//==================================================================================================
//								RJM Maszyny sp. z o.o.
//									13.05.2022
//	Program główny sterujący  
// 	v1.0	|| TC v 3.1.4024.22		|| - pierwsza wersja
//==================================================================================================
PROGRAM MAIN
VAR
	bCzujnik0								: FB_Czujnik_NO;
	bCzujnikMax								: FB_Czujnik_NO;
	fbElektrozawor							: FB_Elektrozawor_5na2_2Cewki;
	fbSilownik								: FB_Silownik_Kontola (fbCzujnikPozycja0 := bCzujnik0, 
																	fbCzujnikPozycjaMax := bCzujnikMax,
																	fbElektrozawor := fbElektrozawor);
	bDoPoczatku: BOOL;
	bDoKonca: BOOL;
	bNaPoczatku: BOOL;
	bNaKoncu: BOOL;


END_VAR

fbSilownik ();
fbSilownik.Praca ();

IF (bDoPoczatku) THEN
	fbSilownik.PrzesunDoPoczatku			:= TRUE;
	bDoPoczatku								:= FALSE;
END_IF

IF (bDoKonca) THEN
	fbSilownik.PrzesunDoKonca				:= TRUE;
	bDoKonca								:= FALSE;
END_IF

bNaPoczatku									:= fbSilownik.NaPoczatku;
bNaKoncu									:= fbSilownik.NaKoncu;

END_PROGRAM

(* stored: Version 1.1.0.1, ProductVersion 3.1.4024.11
   POU MAIN: Id {b8095503-fd65-4541-a4db-ff211f9f14cc}, SpecialFunc None *)
